{attribute 'GeneratedUsingTerminal: EL2911-0000-0016'}
{attribute addProperty BoxType "EL2911-0000-0016"}
{attribute addProperty Id "FSOEAT %I*FSOE_BDDA353211"}
{attribute addProperty CRC "3244414912"}
{attribute addProperty Size "11"}
TYPE FSoE_Inputs_C161D7C0 :
STRUCT
	{attribute addProperty Name "FSOE"}
	FSOE AT %I* : FSOE_BDDA3532;
END_STRUCT
END_TYPE

(* stored: Version 1.2.0.0, ProductVersion 3.1.4024.9
   DUT FSoE_Inputs_C161D7C0: Id {8596f4f0-8860-4ebc-84c2-845e2271b0b6} *)
